PROGRAM MAIN
VAR
	power_OK,
	phase_available,
	ready,
	power_failure,
	error,
	reset, 
	warning : BOOL := FALSE;
	warn_blink : FB_BLINK;
	// TCS remote start;
	remote_start:	BOOL := FALSE;
	// TCS remote stop;
	remote_stop:	BOOL := FALSE;
	power_watchdog : TON;
	ready_state: RS;
	cabinet_temperature:	REAL;
END_VAR

(* 
Main control loop
* Execute sub modules
* power management
* control panel switches and status lamps

* start switch activates Hydraulics and Trafo
* 
*)
power_OK := GVL_main.power_available;
phase_available := GVL_Main.phase_available;

ready_state(SET := power_OK AND HydraulicsControl.oil_pressure_OK AND (GVL_Main.start_switch OR remote_start),
			RESET1 := GVL_main.stop_switch OR remote_stop OR error OR HydraulicsControl.pressure_failure,
			Q1 => ready);
		
TelescopeControl();
DomeControl();
PendantControl();
HydraulicsControl();
GVL_Telescope.brake_azimuth_eve := (GVL_Main.brake_clearing OR PendantControl.brake_open) AND 
									HydraulicsControl.oil_pressure_OK AND 
									NOT GVL_Telescope.azimut_limit_switch;
GVL_Main.softstart_trafo := GVL_Main.key_switch_remote AND NOT power_failure;
power_watchdog(IN := GVL_Main.softstart_trafo AND NOT power_OK,
				PT := T#2S,
				Q => power_failure);
warn_blink(ENABLE := HydraulicsControl.oil_warning, Q => warning);
error := power_failure OR 
			HydraulicsControl.pressure_failure OR 
			(NOT phase_available)
			OR GVL_Telescope.azimut_limit_switch
			OR PendantControl.error
			OR FanControl.error
			OR GVL_Safety.Error;
reset := GVL_Main.reset_switch OR GVL_pendant_control.reset_switch;		
					
GVL_Main.lamp_ready := ready;
GVL_Main.lamp_error := error OR warning;
GVL_Main.lamp_power := power_ok;
cabinet_temperature := INT_TO_REAL(GVL_Main.main_cabinet_temperature) / 100.0;
SafetyHandling();

END_PROGRAM

(* stored: Version 1.1.0.1, ProductVersion 3.1.4024.0
   POU MAIN: Id {c39aef1e-7c14-41dc-ad83-03bececdc52a}, SpecialFunc None *)
